FUNCTION_BLOCK FB_Module_SFC extends FB_Controller_SFC

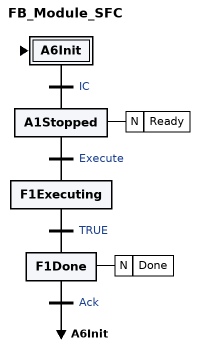
INITIAL_STEP A6Init:
END_STEP
TRANSITION FROM A6Init TO A1Stopped
    := IC;
END_TRANSITION
STEP A1Stopped:
    Ready(N);
END_STEP
TRANSITION FROM A1Stopped TO F1Executing
    := Execute;
END_TRANSITION
STEP F1Executing:
END_STEP
TRANSITION FROM F1Executing TO F1Done
    := TRUE;
END_TRANSITION
STEP F1Done:
    Done(N);
END_STEP
TRANSITION FROM F1Done TO A6Init
    := Ack;
END_TRANSITION

END_FUNCTION_BLOCK

(* stored: Version 1.1.0.1, ProductVersion 3.1.4024.11
   POU FB_Module_SFC: Id {885e2d81-7b5e-4194-aca1-fe47d3a147b8}, SpecialFunc None *)
